ABB RobotStudio station: IRB1600_20220613-165843.rsstn

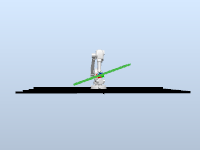
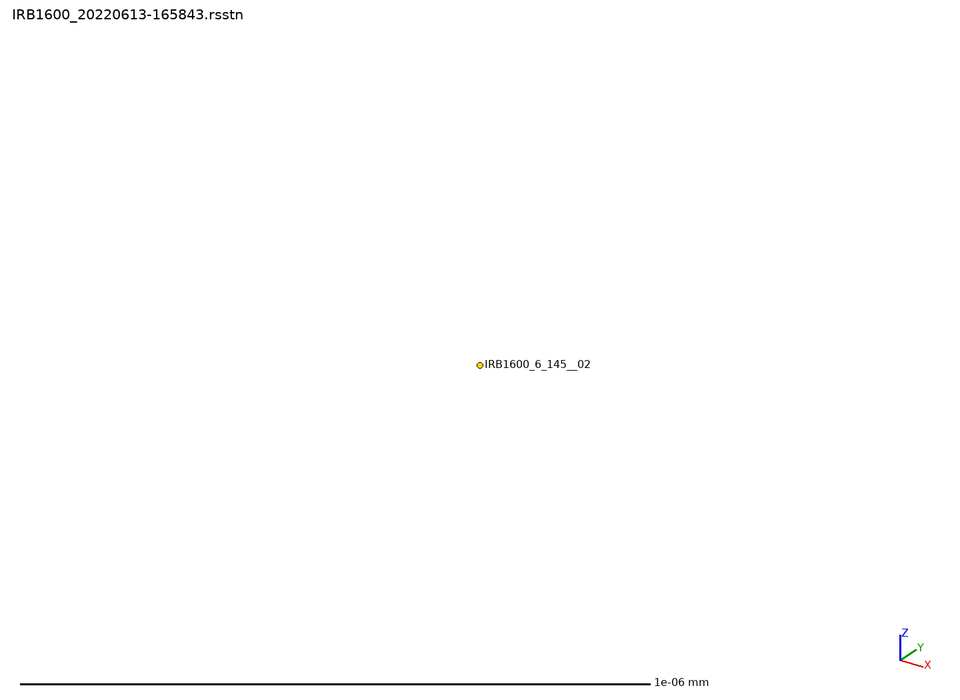
[picture v1: parts stored in the station drawn from their meshes, with robot base, taught points and paths (robot models come from the ABB library and are not in the file)]
Station Solution1 (saved by RobotStudio 21.2.9526.0)
Controller IRB1600_6_145
  mechanical unit ROB_1: IRB1600_6_145__02, 6 joints, base frame (0, 0, 0) mm
Layout (positions relative to the parent item):
  - IRB1600_6_145__02 [mechanism, from Robots\IRB1600_6_145_G_02.rslib] at (0, 0, 0) mm; joint values [-0.0122, 0.7368, 0.5685, -0.0126, -1.3053, 0.3524] (rad or m)
  - surface [part] at (1600, 0, 400) mm, rotated rx 20 ry 0.53 rz 0.19 deg, size 1500 x 1500 x 50 mm
  - flange_connector [part, from Tools\IsoPlate_small_Binzel.rslib] at (842.73, -9.46, 425.99) mm, rotated rx 90 ry 70 rz 90 deg
  - Frame_1 [frame] at (1600, 0, 400) mm, rotated rx 20 ry 0.53 rz 0.19 deg
  - Frame_2 [frame] at (0, 0, 0) mm, rotated rx 0 ry 90 rz 0 deg
Attachment: flange_connector is attached to IRB1600_6_145__02 / Link6
Attachment: Frame_1 is attached to surface
Attachment: surface is attached to flange_connector
Targets, tools, work objects and paths stored in the station, written as RAPID:
! task T_ROB1
MODULE Module1
  LOCAL PERS wobjdata egm_wobj:=[FALSE,TRUE,"",[[0,0,0],[1,0,0,0]],[[0,0,0],[1,0,0,0]]];
  PROC main()
    ConfJ \Off;
    MoveJ RelTool (CRobT(\Tool:=Tooldata_7\wobj:=wobj0), 0, 230, -619.57 \Rx:=-19, \Ry:=10, \Rz:=0),v100,z1,tool0;
    MoveJ RelTool (CRobT(\Tool:=Tooldata_7\wobj:=wobj0), 0, 0, -46.427 \Rx:=-0, \Ry:=-20, \Rz:=0),v100,z1,tool0;
    MoveJ RelTool (CRobT(\Tool:=Tooldata_7\wobj:=wobj0), 0, 0, 46.427 \Rx:=5, \Ry:=-4, \Rz:=0),v100,z1,tool0;
    MoveJ RelTool (CRobT(\Tool:=Tooldata_7\wobj:=wobj0), 0, 0, 73.407 \Rx:=1, \Ry:=14, \Rz:=0),v100,z1,tool0;
    MoveJ RelTool (CRobT(\Tool:=Tooldata_7\wobj:=wobj0), 0, 0, 0 \Rx:=-1, \Ry:=14, \Rz:=0),v100,z1,tool0;
    MoveJ RelTool (CRobT(\Tool:=Tooldata_7\wobj:=wobj0), 0, 0, -73.407 \Rx:=14, \Ry:=-6, \Rz:=0),v100,z1,tool0;
    MoveJ RelTool (CRobT(\Tool:=Tooldata_7\wobj:=wobj0), 0, 0, -32.829 \Rx:=-0, \Ry:=-8, \Rz:=0),v100,z1,tool0;
    MoveJ RelTool (CRobT(\Tool:=Tooldata_7\wobj:=wobj0), 0, 0, 0 \Rx:=-0, \Ry:=-8, \Rz:=0),v100,z1,tool0;
    MoveJ RelTool (CRobT(\Tool:=Tooldata_7\wobj:=wobj0), 0, 0, 32.829 \Rx:=-0, \Ry:=0, \Rz:=0),v100,z1,tool0;
    MoveJ RelTool (CRobT(\Tool:=Tooldata_7\wobj:=wobj0), 0, 0, 32.829 \Rx:=18, \Ry:=8, \Rz:=0),v100,z1,tool0;
    MoveJ RelTool (CRobT(\Tool:=Tooldata_7\wobj:=wobj0), 0, 0, 0 \Rx:=1, \Ry:=-10, \Rz:=0),v100,z1,tool0;
    MoveJ RelTool (CRobT(\Tool:=Tooldata_7\wobj:=wobj0), 0, 0, 46.427 \Rx:=-38, \Ry:=0, \Rz:=0),v100,z1,tool0;
    MoveJ RelTool (CRobT(\Tool:=Tooldata_7\wobj:=wobj0), 0, 0, 46.427 \Rx:=19, \Ry:=2, \Rz:=0),v100,z1,tool0;
    MoveJ RelTool (CRobT(\Tool:=Tooldata_7\wobj:=wobj0), 0, 0, 32.829 \Rx:=-0, \Ry:=0, \Rz:=0),v100,z1,tool0;
    MoveJ RelTool (CRobT(\Tool:=Tooldata_7\wobj:=wobj0), 0, 0, 32.829 \Rx:=-0, \Ry:=8, \Rz:=0),v100,z1,tool0;
    MoveJ RelTool (CRobT(\Tool:=Tooldata_7\wobj:=wobj0), 0, 0, 0 \Rx:=19, \Ry:=-10, \Rz:=0),v100,z1,tool0;
    MoveJ RelTool (CRobT(\Tool:=Tooldata_7\wobj:=wobj0), 0, 0, 46.427 \Rx:=-19, \Ry:=-3, \Rz:=0),v100,z1,tool0;
    MoveJ RelTool (CRobT(\Tool:=Tooldata_7\wobj:=wobj0), 0, 0, 65.657 \Rx:=-0, \Ry:=13, \Rz:=0),v100,z1,tool0;
    MoveJ RelTool (CRobT(\Tool:=Tooldata_7\wobj:=wobj0), 0, 0, 0 \Rx:=19, \Ry:=10, \Rz:=0),v100,z1,tool0;
    MoveJ RelTool (CRobT(\Tool:=Tooldata_7\wobj:=wobj0), 0, 0, -46.427 \Rx:=-0, \Ry:=-20, \Rz:=0),v100,z1,tool0;
    MoveJ RelTool (CRobT(\Tool:=Tooldata_7\wobj:=wobj0), 0, 0, 46.427 \Rx:=-19, \Ry:=-3, \Rz:=0),v100,z1,tool0;
    MoveJ RelTool (CRobT(\Tool:=Tooldata_7\wobj:=wobj0), 0, 0, 65.657 \Rx:=-20, \Ry:=-1, \Rz:=0),v100,z1,tool0;
    MoveJ RelTool (CRobT(\Tool:=Tooldata_7\wobj:=wobj0), 0, 0, 73.407 \Rx:=1, \Ry:=4, \Rz:=0),v100,z1,tool0;
    MoveJ RelTool (CRobT(\Tool:=Tooldata_7\wobj:=wobj0), 0, 0, 46.427 \Rx:=19, \Ry:=2, \Rz:=0),v100,z1,tool0;
    MoveJ RelTool (CRobT(\Tool:=Tooldata_7\wobj:=wobj0), 0, 0, 32.829 \Rx:=-0, \Ry:=0, \Rz:=0),v100,z1,tool0;
    MoveJ RelTool (CRobT(\Tool:=Tooldata_7\wobj:=wobj0), 0, 0, 32.829 \Rx:=-0, \Ry:=-5, \Rz:=0),v100,z1,tool0;
    MoveJ RelTool (CRobT(\Tool:=Tooldata_7\wobj:=wobj0), 0, 0, 65.657 \Rx:=-16, \Ry:=-3, \Rz:=0),v100,z1,tool0;
    MoveJ RelTool (CRobT(\Tool:=Tooldata_7\wobj:=wobj0), 0, 0, 92.853 \Rx:=-2, \Ry:=16, \Rz:=0),v100,z1,tool0;
    MoveJ RelTool (CRobT(\Tool:=Tooldata_7\wobj:=wobj0), 0, 0, 0 \Rx:=-1, \Ry:=-10, \Rz:=0),v100,z1,tool0;
    MoveJ RelTool (CRobT(\Tool:=Tooldata_7\wobj:=wobj0), 0, 0, 46.427 \Rx:=5, \Ry:=-4, \Rz:=0),v100,z1,tool0;
    MoveJ RelTool (CRobT(\Tool:=Tooldata_7\wobj:=wobj0), 0, 0, 73.407 \Rx:=-5, \Ry:=4, \Rz:=0),v100,z1,tool0;
    MoveJ RelTool (CRobT(\Tool:=Tooldata_7\wobj:=wobj0), 0, 0, 46.427 \Rx:=-0, \Ry:=0, \Rz:=0),v100,z1,tool0;
    MoveJ RelTool (CRobT(\Tool:=Tooldata_7\wobj:=wobj0), 0, 0, 46.427 \Rx:=19, \Ry:=10, \Rz:=0),v100,z1,tool0;
    MoveJ RelTool (CRobT(\Tool:=Tooldata_7\wobj:=wobj0), 0, 0, 0 \Rx:=-19, \Ry:=-10, \Rz:=0),v100,z1,tool0;
    MoveJ RelTool (CRobT(\Tool:=Tooldata_7\wobj:=wobj0), 0, 0, 46.427 \Rx:=19, \Ry:=2, \Rz:=0),v100,z1,tool0;
    MoveJ RelTool (CRobT(\Tool:=Tooldata_7\wobj:=wobj0), 0, 0, 32.829 \Rx:=-0, \Ry:=8, \Rz:=0),v100,z1,tool0;
    MoveJ RelTool (CRobT(\Tool:=Tooldata_7\wobj:=wobj0), 0, 0, 0 \Rx:=-18, \Ry:=0, \Rz:=0),v100,z1,tool0;
    MoveJ RelTool (CRobT(\Tool:=Tooldata_7\wobj:=wobj0), 0, 0, 0 \Rx:=-1, \Ry:=-10, \Rz:=0),v100,z1,tool0;
    MoveJ RelTool (CRobT(\Tool:=Tooldata_7\wobj:=wobj0), 0, 0, 46.427 \Rx:=-1, \Ry:=-4, \Rz:=0),v100,z1,tool0;
    MoveJ RelTool (CRobT(\Tool:=Tooldata_7\wobj:=wobj0), 0, 0, 73.407 \Rx:=4, \Ry:=-2, \Rz:=0),v100,z1,tool0;
    MoveJ RelTool (CRobT(\Tool:=Tooldata_7\wobj:=wobj0), 0, 0, 92.853 \Rx:=2, \Ry:=30, \Rz:=0),v100,z1,tool0;
    MoveJ RelTool (CRobT(\Tool:=Tooldata_7\wobj:=wobj0), 0, 0, -73.407 \Rx:=-6, \Ry:=0, \Rz:=0),v100,z1,tool0;
    MoveJ RelTool (CRobT(\Tool:=Tooldata_7\wobj:=wobj0), 0, 0, -73.407 \Rx:=20, \Ry:=-14, \Rz:=0),v100,z1,tool0;
    MoveJ RelTool (CRobT(\Tool:=Tooldata_7\wobj:=wobj0), 0, 0, 0 \Rx:=-0, \Ry:=-8, \Rz:=0),v100,z1,tool0;
    MoveJ RelTool (CRobT(\Tool:=Tooldata_7\wobj:=wobj0), 0, 0, 32.829 \Rx:=-0, \Ry:=-5, \Rz:=0),v100,z1,tool0;
    MoveJ RelTool (CRobT(\Tool:=Tooldata_7\wobj:=wobj0), 0, 0, 65.657 \Rx:=-19, \Ry:=3, \Rz:=0),v100,z1,tool0;
    MoveJ RelTool (CRobT(\Tool:=Tooldata_7\wobj:=wobj0), 0, 0, 46.427 \Rx:=-0, \Ry:=0, \Rz:=0),v100,z1,tool0;
    MoveJ RelTool (CRobT(\Tool:=Tooldata_7\wobj:=wobj0), 0, 0, 46.427 \Rx:=19, \Ry:=2, \Rz:=0),v100,z1,tool0;
    MoveJ RelTool (CRobT(\Tool:=Tooldata_7\wobj:=wobj0), 0, 0, 32.829 \Rx:=-18, \Ry:=8, \Rz:=0),v100,z1,tool0;
    MoveJ RelTool (CRobT(\Tool:=Tooldata_7\wobj:=wobj0), 0, 0, 0 \Rx:=-1, \Ry:=-10, \Rz:=0),v100,z1,tool0;
    MoveJ RelTool (CRobT(\Tool:=Tooldata_7\wobj:=wobj0), 0, 0, 46.427 \Rx:=-0, \Ry:=0, \Rz:=0),v100,z1,tool0;
    MoveJ RelTool (CRobT(\Tool:=Tooldata_7\wobj:=wobj0), 0, 0, 46.427 \Rx:=19, \Ry:=10, \Rz:=0),v100,z1,tool0;
    MoveJ RelTool (CRobT(\Tool:=Tooldata_7\wobj:=wobj0), 0, 0, 0 \Rx:=-0, \Ry:=-8, \Rz:=0),v100,z1,tool0;
    MoveJ RelTool (CRobT(\Tool:=Tooldata_7\wobj:=wobj0), 0, 0, 32.829 \Rx:=-0, \Ry:=0, \Rz:=0),v100,z1,tool0;
    MoveJ RelTool (CRobT(\Tool:=Tooldata_7\wobj:=wobj0), 0, 0, 32.829 \Rx:=-0, \Ry:=16, \Rz:=0),v100,z1,tool0;
  ENDPROC
  PROC EGM_CARTESIAN_MOVE()
    WaitTime 2;
  ENDPROC
  PROC RAPID_MOVE()
  ENDPROC
ENDMODULE

! task T_ROB1
MODULE CalibData
  TASK PERS tooldata Tooldata_4:=[TRUE,[[0,0,0],[1,0,0,0]],[1,[0,0,1],[1,0,0,0],0,0,0]];
  TASK PERS tooldata Tooldata_5:=[TRUE,[[0,0,0],[1,0,0,0]],[1,[0,0,1],[1,0,0,0],0,0,0]];
  TASK PERS tooldata Tooldata_6:=[TRUE,[[0,0,0],[1,0,0,0]],[1,[0,0,1],[1,0,0,0],0,0,0]];
  TASK PERS tooldata Tooldata_7:=[TRUE,[[27.654,0,757.266],[0.707106781,0,-0.707106781,0]],[1,[0,0,1],[1,0,0,0],0,0,0]];
ENDMODULE

